FUNCTION_BLOCK FB_Axis
VAR_INPUT
	
	sAXIS_STATE:STRING:='UNINIT';
	sName:STRING;
	Axis:Axis_ref;
	bEnable:BOOL:=FALSE;
	bHalt:BOOL:=FALSE;
	bHOME:BOOL:=FALSE;
	bHOME_DIR:BOOL;
	bReset:BOOL:=FALSE;
	bSetPosition:BOOL:=FALSE;
	Dist:REAL;
	bMoveRel:BOOL:=FALSE;
	bMoveRelBusy:BOOL;
	rPos:LREAL;
	rVel:LREAL:=20;
	rAcc:LREAL;
	rDec:LREAL;
	rJerk:LREAL;
	bMoveABS:BOOL:=FALSE;
	bMoveAbsBusy:BOOL;
	bJogPos:BOOL;
	bJogNeg:BOOL;
	bMANUAL:BOOL:=FALSE;
	tACTION:TON;
	ton_Reset: TON;
	bOPEN:BOOL;
	bCLOSE:BOOL;
	bLIMIT_OPENED:BOOL;
	bLIMIT_CLOSED:BOOL;
	bLIMIT:BOOL;
	rACTION_TIMEOUT:TIME:=T#10S;
	jogVEL: REAL;
	jogHOME_VEL: REAL;
	jogOPEN_VEL: REAL;
	jogCLOSE_VEL: REAL;
	bSTOP:BOOL;
	bSTOP_ALL:BOOL;
END_VAR

VAR_OUTPUT
	bOPENED:BOOL;
	bCLOSED:BOOL;
	bHOMED:BOOL;
	bBusy: BOOL;
	bAXIS_ERROR:BOOL;
	bSTATE_ERROR:BOOL;
	bInPos:BOOL;
	rActPos:LREAL;
	rActVel:LREAL;
	bRelDone:BOOL;
	bAbsDone:BOOL;
	bHaltDone:BOOL;
	bNOT_ENABLE:BOOL;
END_VAR
VAR
	bSTART_ACTION:BOOL;
	iHOME_STATE: INT:=98;
	iAXIS_STATE:INT:=98;
	tDelay: TON;
	bDelay:BOOL:=FALSE;
	MoveAbsolute: MC_MoveAbsolute;
	power: MC_Power;
	Reset: MC_Reset;
	SetPosition: MC_SetPosition;
	JOG: MC_Jog;
	RELATIVE: MC_MoveRelative;
	HALT: MC_Halt;
	HOME: MC_Home;
	bFirst_run:BOOL:=FALSE;
	bStopBusy:BOOL;
	
	
	
	
END_VAR

IF NOT bFirst_run THEN
	RESET.Execute:=TRUE;
	 bFirst_run:=TRUE;
END_IF
bNOT_ENABLE:=NOT bENABLE;
rActPos:=Axis.NcToPlc.ActPos;
rActVel:=Axis.NcToPlc.ActVelo;



IF RELATIVE.Busy OR JOG.Busy OR moveAbsolute.busy THEN
	bBusy:=TRUE;
	bHOMED:=FALSE;
END_IF
IF NOT RELATIVE.Busy AND NOT JOG.Busy AND NOT moveAbsolute.busy THEN
	bBusy:=FALSE;
END_IF

IF POWER.error OR RELATIVE.error OR MoveAbsolute.error OR JOG.error THEN
	bAXIS_ERROR:=TRUE;
END_IF
IF NOT POWER.error AND NOT RELATIVE.error AND NOT MoveAbsolute.error AND NOT JOG.error THEN
	bAXIS_ERROR:=FALSE;
END_IF

IF bRelDone OR  bAbsDone THEN
	bInPos:=TRUE;
END_IF
IF bBusy THEN
	bInPos:=FALSE;
	bRelDone:=FALSE;
	bAbsDone:=FALSE;
END_IF


CMDs();
mAXIS_STATE_MACHINE();

ACTION aAXIS_ERROR:
gEventType:= 'axis Alarm'; 
gEventSeverity:= 'Error';

gEventName:= sNAME;
IF iAXIS_STATE=1  THEN
	gEventText:='axis homing';
	gEventIdentity:=2001;
END_IF
IF iAXIS_STATE=20  THEN
	gEventText:='axis opening';
	gEventIdentity:=2002;
END_IF
IF iAXIS_STATE=40  THEN
	gEventText:='axis closing';
	gEventIdentity:=2003;
END_IF
fbEventLogger.mAdd();
END_ACTION

METHOD clear_cmd_req : BOOL
VAR_INPUT
END_VAR

bMoveABS:= bMoveRel:= bJogPos:= bJogNeg:=FALSE;
END_METHOD

ACTION CMDs:
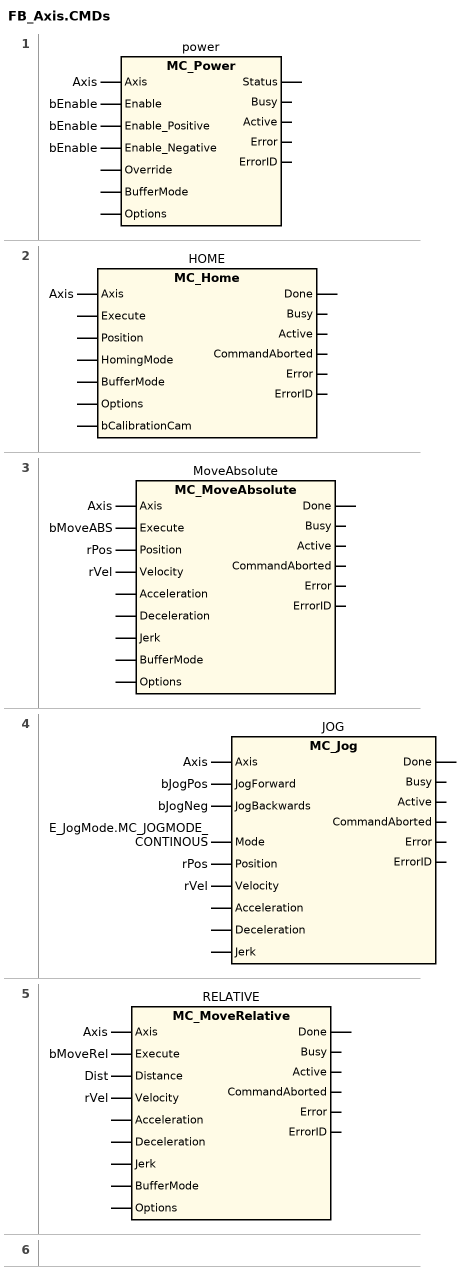
// NETWORK 1
power(Axis := Axis, Enable := bEnable, Enable_Positive := bEnable, Enable_Negative := bEnable); // MC_Power

// NETWORK 2
HOME(Axis := Axis); // MC_Home

// NETWORK 3
MoveAbsolute(Axis := Axis, Execute := bMoveABS, Position := rPos, Velocity := rVel); // MC_MoveAbsolute

// NETWORK 4
JOG(
    Axis := Axis,
    JogForward := bJogPos,
    JogBackwards := bJogNeg,
    Mode := E_JogMode.MC_JOGMODE_CONTINOUS,
    Position := rPos,
    Velocity := rVel); // MC_Jog

// NETWORK 5
RELATIVE(Axis := Axis, Execute := bMoveRel, Distance := Dist, Velocity := rVel); // MC_MoveRelative

// NETWORK 6

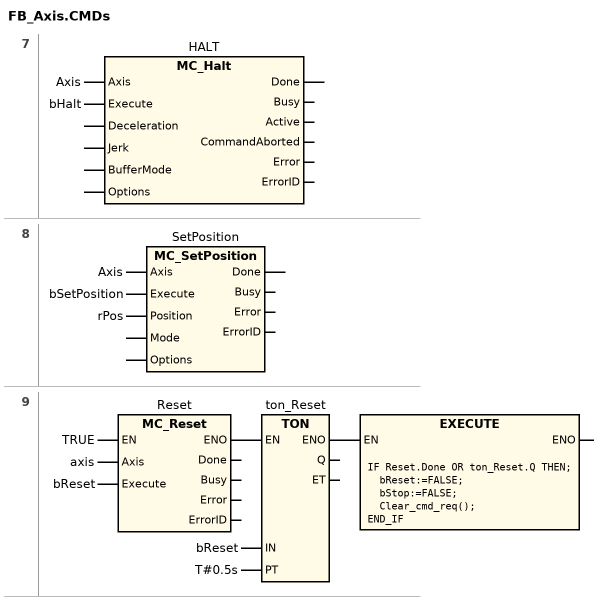
// NETWORK 7
HALT(Axis := Axis, Execute := bHalt); // MC_Halt

// NETWORK 8
SetPosition(Axis := Axis, Execute := bSetPosition, Position := rPos); // MC_SetPosition

// NETWORK 9
Reset(Axis := axis, Execute := bReset); // MC_Reset
ton_Reset(IN := bReset, PT := T#0.5s); // TON

IF Reset.Done OR ton_Reset.Q THEN;
	bReset:=FALSE;
	bStop:=FALSE;
	Clear_cmd_req();
END_IF
END_ACTION

METHOD mAXIS_STATE_MACHINE : BOOL
VAR_INPUT
	
END_VAR
tACTION(IN:= bSTART_ACTION, PT:=rACTION_TIMEOUT , Q=> , ET=> );
IF bHOME_DIR THEN
	bLIMIT:=bLIMIT_OPENED;
ELSE
	bLIMIT:=bLIMIT_CLOSED;
END_IF

IF bSTOP_ALL THEN
	iAXIS_STATE:=99;
	bSTOP_ALL:=FALSE;
	bSTART_ACTION:=FALSE;
END_IF

CASE iAXIS_STATE OF
	1:// ============================================== HOMING
		bSTART_ACTION:=TRUE;
		sAXIS_STATE:='HOMING - TO SENSOR';
		bOPENED:=FALSE;bCLOSED:=FALSE;bOPEN:=FALSE;bCLOSE:=FALSE;bHOMED:=FALSE;bHOME:=FALSE;
		bENABLE:=TRUE;
		rVel:= jogHOME_VEL;
		IF bHOME_DIR THEN
			bJogPos:=TRUE;
		ELSE
			bJogNeg:=TRUE;
		END_IF
		
		IF bLIMIT THEN
			bSTART_ACTION:=FALSE;
			bJogNeg:=FALSE;
			bJogPos:=FALSE;
			iAXIS_STATE:=2;
		END_IF
		IF tACTION.Q THEN
			bSTART_ACTION:=FALSE;
			aAXIS_ERROR();
			iAXIS_STATE:=99;
			bSTATE_ERROR:=TRUE;
		END_IF
	2://FROM LIMIT
			sAXIS_STATE:= 'HOMING- FROM SENSOR';
			IF Axis.NcToPlc.ActVelo= 0 THEN
				
				//rVel:= 3;
				//IF bHOME_DIR THEN
				//	bJogNeg:=TRUE;
				//ELSE
					//bJogPos:=TRUE;
				//END_IF
				iAXIS_STATE:=3;
			END_IF	
	3:// FINISH
			//IF NOT bLIMIT THEN
				//bJogNeg:=FALSE;
				//bJogPos:=FALSE;
				IF Axis.NcToPlc.ActVelo= 0 THEN
					bHOMED:=TRUE;
					IF bHOME_DIR THEN
						iAXIS_STATE:=100;// to ready state
						bOPENED:=TRUE;
					ELSE
						iAXIS_STATE:=100;// to ready state
						bCLOSED:=TRUE;
					END_IF
				END_IF
			//END_IF
	20://=============================================== OPENING
		sAXIS_STATE:= 'OPENING';
		bSTART_ACTION:=TRUE;
		bOPENED:=FALSE;bCLOSED:=FALSE;bOPEN:=FALSE;bCLOSE:=FALSE;bHOMED:=FALSE;bHOME:=FALSE;
		bENABLE:=TRUE;
		rVel:= jogOPEN_VEL;
		bJogPos:=TRUE;
		IF bLIMIT_OPENED THEN
			iAXIS_STATE:=21;// to deccell
			bJogPos:=FALSE;
			bSTART_ACTION:=FALSE;
		END_IF
		IF tACTION.Q THEN
			bSTART_ACTION:=FALSE;
			aAXIS_ERROR();
			iAXIS_STATE:=99;
			bSTATE_ERROR:=TRUE;
		END_IF
		
		21:
			sAXIS_STATE:= 'OPEN DECCELERATING';
			IF Axis.NcToPlc.ActVelo=0 THEN
				bENABLE:=FALSE;//////////////////////
				iAXIS_STATE:=100;
				bOPENED:=TRUE;
			END_IF
	
	40://=============================================== CLOSING
		sAXIS_STATE:= 'CLOSING';
		bSTART_ACTION:=TRUE;
		bOPENED:=FALSE;bCLOSED:=FALSE;bOPEN:=FALSE;bCLOSE:=FALSE;bHOMED:=FALSE;bHOME:=FALSE;
		bENABLE:=TRUE;
		rVel:= jogCLOSE_VEL;
		bJogNeg:=TRUE;
		IF bLIMIT_CLOSED THEN
			iAXIS_STATE:=41;// to deccell
			bJogNeg:=FALSE;
			bSTART_ACTION:=FALSE;
		END_IF
		IF tACTION.Q THEN
			bSTART_ACTION:=FALSE;
			aAXIS_ERROR();
			iAXIS_STATE:=99;
			bSTATE_ERROR:=TRUE;
		END_IF
		
		41:
			sAXIS_STATE:= 'CLOSE DECCELERATING';
			IF Axis.NcToPlc.ActVelo=0 THEN
				bENABLE:=FALSE;//////////////////////
				iAXIS_STATE:=100;
				bCLOSED:=TRUE;
			END_IF
	
	50:	//========================ABSOLUTE=====================
	sAXIS_STATE:='MOVING ABSOLUTE';
	bAbsDone:=FALSE; bOPENED:=FALSE;bCLOSED:=FALSE;bOPEN:=FALSE;bCLOSE:=FALSE;bHOMED:=FALSE;bHOME:=FALSE;
	IF moveAbsolute.Done OR HALT.Done THEN
		iAXIS_STATE:=100;
		bAbsDone:=TRUE;
		bMoveAbs:=FALSE;
	END_IF
	51://========================RELATIVE=====================
	sAXIS_STATE:='MOVING RELATIVE';
	bRelDone:=FALSE; bOPENED:=FALSE;bCLOSED:=FALSE;bOPEN:=FALSE;bCLOSE:=FALSE;bHOMED:=FALSE;bHOME:=FALSE;
	IF RELATIVE.Done OR HALT.Done THEN
		iAXIS_STATE:=100; 
		bRelDone:=TRUE;
		bMoveRel:=FALSE;
	END_IF
	52://======================= HALT =========================
	sAXIS_STATE:='HALTING';
	bHaltDone:=FALSE;bOPENED:=FALSE;bCLOSED:=FALSE;bOPEN:=FALSE;bCLOSE:=FALSE;bHOMED:=FALSE;bHOME:=FALSE;
	IF HALT.Done THEN
		iAXIS_STATE:=100;
		bHaltDone:=TRUE;
		bHALT:=FALSE;
	END_IF		
	98:// ============================================ UNINIT
		sAXIS_STATE:='UNINIT';
		IF bHOME THEN
			iAXIS_STATE:=1;
			bSTATE_ERROR:=FALSE;
		END_IF
		
	99://======================================= ERROR 
		sAXIS_STATE:='AXIS STATE ERROR';
		bJogNeg:=FALSE;
		bJogPos:=FALSE;
		bHOMED:=FALSE;
		bNOT_ENABLE:=TRUE;
		clear_cmd_req();
		IF bHOME THEN
			iAXIS_STATE:=1;
			bSTATE_ERROR:=FALSE;
		END_IF
		
	100://=============================================== READY
		sAXIS_STATE:='READY';
		IF bOPENED THEN
		sAXIS_STATE:= 'OPENED';
		END_IF
		IF bCLOSED THEN
		sAXIS_STATE:= 'CLOSED';
		END_IF
		IF bHOME AND NOT bHOMED THEN
			iAXIS_STATE:=1;
			bSTATE_ERROR:=FALSE;
		END_IF
		IF bCLOSE AND NOT bCLOSED THEN
			iAXIS_STATE:=40;
			bSTATE_ERROR:=FALSE;
		END_IF
		IF bOPEN AND NOT bOPENED THEN
			iAXIS_STATE:=20;
			bSTATE_ERROR:=FALSE;
		END_IF
		IF bMoveAbs THEN
			iAXIS_STATE:=50;
			bSTATE_ERROR:=FALSE;
		END_IF
		IF bMoveRel THEN
			iAXIS_STATE:=51;
			bSTATE_ERROR:=FALSE;
		END_IF
		IF bHALT THEN
			iAXIS_STATE:=52;
			bSTATE_ERROR:=FALSE;
		END_IF
	
END_CASE
END_METHOD

END_FUNCTION_BLOCK

(* stored: Version 1.1.0.1, ProductVersion 3.1.4024.12
   POU FB_Axis: Id {1ec8daca-b967-496e-b296-4221933406bb}, SpecialFunc None
   Action aAXIS_ERROR: Id {d9bff058-7cd6-4042-808e-812c3696c258}
   Method clear_cmd_req: Id {c115c33f-8377-4dd1-8142-a1b93e7b6e59}
   Action CMDs: Id {3d4245d8-d06e-4f79-a793-3fc083bab546}
   Method mAXIS_STATE_MACHINE: Id {5855ed75-8fcd-47ee-ae72-6d0b401eafef} *)
